Staubli VAL3: remGetMaxRV.pgx

program remGetMaxRV(string& sReturn[] (dimensions=1))
  local string sCmd
begin
  // Return maximum allowed rotational velocity in deg/s for remote moves.
  //
  logMsg("call remGetMaxRV")
  sCmd="GETMAXRV"
  call remGetnGlobal(nMaxAccel,sCmd,sReturn)
end
